// TwinCAT 3 PLC project PLC1
// ProgramVersion: 3.1.4023.0
// libraries:
//   Tc2_Standard, * (Beckhoff Automation GmbH)
//   Tc2_System, * (Beckhoff Automation GmbH)
//   Tc3_Module, * (Beckhoff Automation GmbH)
// project tree:
//   / PlcTask.TcTTO
//   POUs/ MAIN.TcPOU
// real-time tasks:
//   TASK PlcTask: cycle T#10ms, priority 20, ADS port 350

CONFIGURATION PLC1
    RESOURCE PLC ON TwinCAT3
        TASK PlcTask(INTERVAL := T#10ms, PRIORITY := 20);
        PROGRAM MAIN WITH PlcTask : MAIN;
    END_RESOURCE
END_CONFIGURATION

// ---- POUs/MAIN.TcPOU
PROGRAM MAIN
VAR
	fSin		: REAL;
	fTheta		: REAL := -3.14;
	fbSampling	: TON;
END_VAR

fbSampling(In:=TRUE, PT:=T#1S);

IF fbSampling.Q THEN
	IF fTheta >= 3.14 THEN
		fTheta := -3.14;
	END_IF
	fSin := SIN(fTheta);
	fTheta := fTheta + 0.01;
	fbSampling(In:=FALSE);
END_IF

END_PROGRAM
